FUNCTION_BLOCK STRUCT_DEMUX (* Generic block for demuxing structs *)
  (* Standard: 61499-2; Description: Copyright (c) 2020 Johannes Kepler University Linz This program and the accompanying materials are made available under the terms of the Eclipse Public License 2.0 which is available at https://www.eclipse.org/legal/epl-2.0/ SPDX-License-Identifier: EPL-2.0 *)
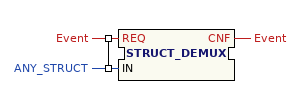
  EVENT_INPUT
    REQ WITH IN; (* Normal Execution Request *)
  END_EVENT
  EVENT_OUTPUT
    CNF; (* Execution Confirmation *)
  END_EVENT
  VAR_INPUT
    IN : ANY_STRUCT;
  END_VAR
  ALGORITHM REQ IN AnyText:

  END_ALGORITHM
END_FUNCTION_BLOCK
